FUNCTION_BLOCK AngularVelocity EXTENDS SM_AngularVelocity
VAR_INPUT
END_VAR
VAR_OUTPUT
END_VAR
VAR
    _testVar : INT;
END_VAR

SUPER^();

END_FUNCTION_BLOCK

(* stored: Version 1.1.0.1, ProductVersion 3.1.4018.5
   POU AngularVelocity: Id {08c034e3-63ab-4bd5-87b5-ac1d75d97172}, SpecialFunc None *)
